// Mitsubishi GX Works2 project: or_2_inputs   PLC: Q03UDV
// LRI_2023

PROGRAM MAIN
VAR
  MO : BOOL;
END_VAR
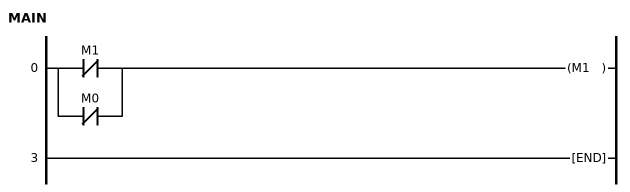
0     LDI     M1
      ORI     M0
      OUT     M1
3     END
END_PROGRAM
